Staubli VAL3: Day13.pjx

--- Day13.pjx ---
Parameters version=s8.13.1Cs9_BS2800 stackSize=5000 millimeterUnit=true
Program file=fold.pgx
Program file=start.pgx
Program file=stop.pgx
Data file=Day13.dtx
Library alias=util path=Disk://helpers/helpers.pjx
Library alias=math path=Disk://math/math.pjx
Library alias=str path=Disk://string/string.pjx
Library alias=stat path=Disk://statistics/statistics.pjx
Library alias=mat path=Disk://matrix/matrix.pjx
Type name=lists path=Disk://types/lists/lists.pjx

--- Day13.dtx ---
string sInput
lists lResult
  [0]
    string sString
num nResult
num nXcoord
num nYcoord
num nFolds
string sFolds
string sGrid
string sResult
num nFolds_
num nGrid[1 1]
num nLeftMatrix[1 1]
num nRightMatrix[1 1]
num nRowSum

--- start.pgx ---
program start()
  local num l_nElement
  local bool l_bBool
  local num l_nXMax
  local num l_nYMax
  local bool l_bFolds
  local num l_nFoldCounter
begin

  // read file
  call util:readFile("Disk://input_day13.txt", sInput)

  // find empty line and devide between grid and folds
  l_bFolds = false
  l_nFoldCounter = 0
  for l_nElement = 0 to size(sInput)-1
    if sInput[l_nElement] == ""
      l_bFolds = true
    endIf
    if l_bFolds
      append(sFolds)
      l_nFoldCounter = l_nFoldCounter+1
      sFolds[l_nFoldCounter] = sInput[l_nElement]
    else
      append(sGrid)
      sGrid[l_nElement+1] = sInput[l_nElement]
    endIf

  endFor

  // delete empty entries
  delete(sGrid[0])
  delete(sFolds[1])
  delete(sFolds[0])

  // get coordinates from sGrid
  call str:splitString(sGrid,",", lResult)

  // prepare coordinates
  resize(nXcoord, 1, size(lResult))
  resize(nYcoord, 1, size(lResult))

  // convert string from coordintes to num
  for l_nElement = 0 to size(lResult)-1
    toNum(lResult[l_nElement].sString[0],nXcoord[l_nElement], l_bBool)
    toNum(lResult[l_nElement].sString[1],nYcoord[l_nElement], l_bBool)
  endFor

  // split folds
  call str:replacePattern(sFolds, "fold along ", "", sResult)
  call str:splitString(sResult, "=", lResult)

  // extract folds
  resize(sFolds, 1, size(lResult))
  resize(nFolds, 1, size(lResult))
  l_nXMax = l_nYMax = 0
  for l_nElement = 0 to size(lResult)-1
    sFolds[l_nElement] = lResult[l_nElement].sString[0]
    call util:vec2num(lResult[l_nElement].sString[1], nFolds_)
    nFolds[l_nElement] = nFolds_
    if sFolds[l_nElement] == "x"
      l_nXMax = max(l_nXMax, nFolds_)
    else
      l_nYMax = max(l_nYMax, nFolds_)
    endIf

  endFor

  // prepare grid
  resize(nGrid,1,l_nXMax*2+1)
  resize(nGrid,2,l_nYMax*2+1)

  for l_nElement = 0 to size(nXcoord)-1
    nGrid[nXcoord[l_nElement], nYcoord[l_nElement]] = 1
  endFor

  // PUZZLE 1: just fold one time
  call fold(sFolds[0], nFolds[0])

  nRowSum = 0
  call util:rowSum(nGrid, nRowSum)
  call math:sum(nRowSum, nResult)
  call util:printNum(nResult)
  // 687


  // Puzzle 2
  // prepare grid
  resize(nGrid,1,l_nXMax*2+1)
  resize(nGrid,2,l_nYMax*2+1)

  for l_nElement = 0 to size(nXcoord)-1
    nGrid[nXcoord[l_nElement], nYcoord[l_nElement]] = 1
  endFor

  for l_nElement = 0 to size(nFolds)-1
    call fold(sFolds[l_nElement], nFolds[l_nElement])
  endFor

  call util:printNum2d(nGrid)
  // FGKCKBZG


end

--- fold.pgx ---
program fold(string x_sDirection, num x_nEdge)
  local num l_nDim[2]
begin

  if x_sDirection == "x"
    // 0123456 7 891011121314
    call util:extractGrid(nGrid,1,0,x_nEdge-1, nLeftMatrix)
    call util:extractGrid(nGrid,1,size(nGrid,1)-1,x_nEdge+1, nRightMatrix)
  else
    call util:extractGrid(nGrid,2,0,x_nEdge-1, nLeftMatrix)
    call util:extractGrid(nGrid,2,size(nGrid,2)-1,x_nEdge+1, nRightMatrix)
  endIf

  call mat:add(nLeftMatrix, nRightMatrix, nGrid)

  // Set to one, if addition will give results > 1
  for l_nDim[0] = 0 to size(nGrid,1)-1
    for l_nDim[1] = 0 to size(nGrid,2) -1
      if nGrid[l_nDim[0], l_nDim[1]] > 1
        nGrid[l_nDim[0], l_nDim[1]] = 1
      endIf
    endFor
  endFor


end
